TYPE ST_ShiftRowV3 :
STRUCT
    StartMin : DINT := -1;
    DurationMin : DINT := 1440;
    ActiveDays : DINT;
    ProductionTarget : DINT;
END_STRUCT
END_TYPE

(* stored: Version 1.1.0.1, ProductVersion 3.1.4024.12
   DUT ST_ShiftRowV3: Id {c87ebe61-537f-4a3c-ae4c-c44a36fba35e} *)
